// Mitsubishi GX Works2 project: ror_rorEx03   PLC: Q02/Q02H

PROGRAM MAIN
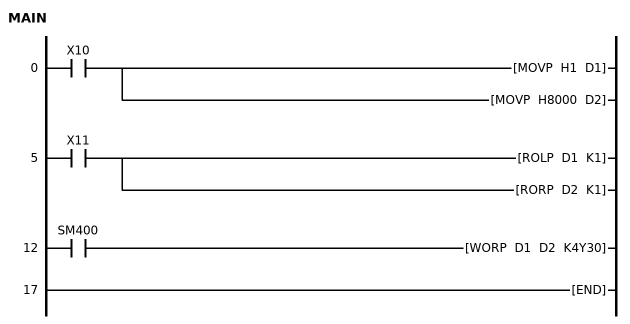
0     LD      X10
      MOVP    H1 D1
      MOVP    H8000 D2
5     LD      X11
      ROLP    D1 K1
      RORP    D2 K1
12    LD      SM400
      WORP    D1 D2 K4Y30
17    END
END_PROGRAM
